FUNCTION_BLOCK Raspador_Gordura (* Composite Function Block Type *)
  (* Standard: 61499-2 *)
  (* Version 0.0, 04/03/2026, template *)
  PACKAGE Hidryco.HidrycoLib;
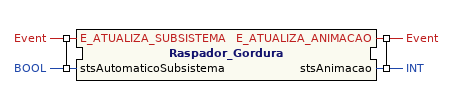
  EVENT_INPUT
    E_ATUALIZA_SUBSISTEMA WITH stsAutomaticoSubsistema;
  END_EVENT
  EVENT_OUTPUT
    E_ATUALIZA_ANIMACAO WITH stsAnimacao;
  END_EVENT
  VAR_INPUT
    stsAutomaticoSubsistema : BOOL;
  END_VAR
  VAR_OUTPUT
    stsAnimacao : INT;
  END_VAR
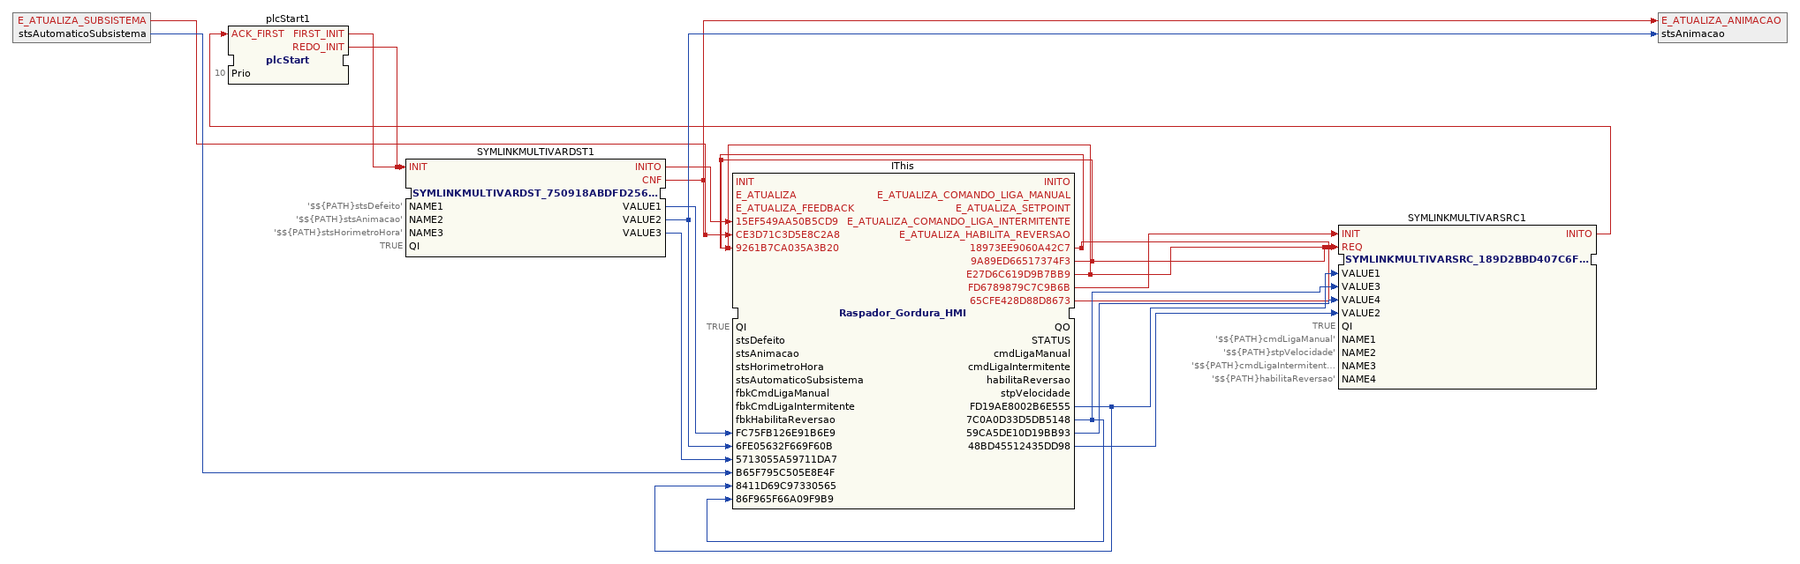
  FBS
    SYMLINKMULTIVARDST1 : SYMLINKMULTIVARDST_750918ABDFD25675(NAME1 := '$${PATH}stsDefeito', NAME2 := '$${PATH}stsAnimacao', NAME3 := '$${PATH}stsHorimetroHora', QI := TRUE); {SET_ATTRIBUTE(Configuration.GenericFBType.InterfaceParams, Runtime.System#I:=3;VALUE${I$}:BOOL,INT,DINT)}
    IThis : Raspador_Gordura_HMI(QI := TRUE);
    SYMLINKMULTIVARSRC1 : SYMLINKMULTIVARSRC_189D2BBD407C6F124(QI := TRUE, NAME1 := '$${PATH}cmdLigaManual', NAME2 := '$${PATH}stpVelocidade', NAME3 := '$${PATH}cmdLigaIntermitente', NAME4 := '$${PATH}habilitaReversao'); {SET_ATTRIBUTE(Configuration.GenericFBType.InterfaceParams, Runtime.System#I:=4;VALUE${I$}:BOOL,INT,BOOL,BOOL)}
    plcStart1 : plcStart(Prio := 10);
  END_FBS
  EVENT_CONNECTIONS
    plcStart1.FIRST_INIT TO SYMLINKMULTIVARDST1.INIT;
    plcStart1.REDO_INIT TO SYMLINKMULTIVARDST1.INIT;
    SYMLINKMULTIVARSRC1.INITO TO plcStart1.ACK_FIRST;
    SYMLINKMULTIVARDST1.INITO TO IThis.15EF549AA50B5CD9;
    SYMLINKMULTIVARDST1.CNF TO IThis.CE3D71C3D5E8C2A8;
    IThis.18973EE9060A42C7 TO IThis.9261B7CA035A3B20;
    IThis.9A89ED66517374F3 TO IThis.9261B7CA035A3B20;
    IThis.E27D6C619D9B7BB9 TO IThis.9261B7CA035A3B20;
    IThis.FD6789879C7C9B6B TO SYMLINKMULTIVARSRC1.INIT;
    IThis.E27D6C619D9B7BB9 TO SYMLINKMULTIVARSRC1.REQ;
    IThis.65CFE428D88D8673 TO SYMLINKMULTIVARSRC1.REQ;
    IThis.18973EE9060A42C7 TO SYMLINKMULTIVARSRC1.REQ;
    IThis.9A89ED66517374F3 TO SYMLINKMULTIVARSRC1.REQ;
    E_ATUALIZA_SUBSISTEMA TO IThis.CE3D71C3D5E8C2A8;
    SYMLINKMULTIVARDST1.CNF TO E_ATUALIZA_ANIMACAO;
  END_CONNECTIONS
  DATA_CONNECTIONS
    SYMLINKMULTIVARDST1.VALUE1 TO IThis.FC75FB126E91B6E9;
    SYMLINKMULTIVARDST1.VALUE2 TO IThis.6FE05632F669F60B;
    SYMLINKMULTIVARDST1.VALUE3 TO IThis.5713055A59711DA7;
    stsAutomaticoSubsistema TO IThis.B65F795C505E8E4F;
    IThis.FD19AE8002B6E555 TO IThis.8411D69C97330565;
    IThis.7C0A0D33D5DB5148 TO IThis.86F965F66A09F9B9;
    IThis.FD19AE8002B6E555 TO SYMLINKMULTIVARSRC1.VALUE1;
    IThis.7C0A0D33D5DB5148 TO SYMLINKMULTIVARSRC1.VALUE3;
    IThis.59CA5DE10D19BB93 TO SYMLINKMULTIVARSRC1.VALUE4;
    IThis.48BD45512435DD98 TO SYMLINKMULTIVARSRC1.VALUE2;
    SYMLINKMULTIVARDST1.VALUE2 TO stsAnimacao;
  END_CONNECTIONS
END_FUNCTION_BLOCK
